{attribute 'qualified_only'}
VAR_GLOBAL
    {attribute 'pytmc' := 'pv: PLC:LFE:MOTION:ARB'}
    fbArbiter: FB_Arbiter(1);

    {attribute 'pytmc' := 'pv: PLC:LFE:MOTION:FFO:01'}
    {attribute 'TcLinkTo' := '.q_xFastFaultOut:=TIIB[PMPS_FFO]^Channel 1^Output'}
    fbFastFaultOutput1: FB_HardwareFFOutput := (bAutoReset := TRUE, i_sNetID := '172.21.88.66.1.1');

    {attribute 'pytmc' := 'pv: PLC:LFE:MOTION:FFO:02'}
    {attribute 'TcLinkTo' := '.q_xFastFaultOut:=TIIB[PMPS_FFO]^Channel 2^Output'}
    fbFastFaultOutput2: FB_HardwareFFOutput := (bAutoReset := TRUE, i_sNetID := '172.21.88.66.1.1');

    {attribute 'pytmc' := 'pv: PLC:LFE:MOTION:PMPS:ReqTrans'}
    rReqTrans AT %I*		: ARRAY [1..PMPS_GVL.AUX_ATTENUATORS] OF ST_PMPS_Attenuator_IO;
    {attribute 'pytmc' := 'pv: PLC:LFE:MOTION:PMPS:CurTrans'}
    rCurTrans AT %Q*		: ARRAY [1..PMPS_GVL.AUX_ATTENUATORS] OF ST_PMPS_Attenuator_IO;

    ePF1L0State: E_WFS_States;
END_VAR

(* stored: Version 1.1.0.1
   GVL GVL: Id {7ed09a37-cf90-49ac-9e4a-5fe59e47274f} *)
